INTERFACE I_NodePrototypes EXTENDS I_Serializable

METHOD PUBLIC InsertByType
VAR_INPUT
	NodeType : T_MAXSTRING;
	NodePrototype : I_NodePrototype;
END_VAR
END_METHOD

METHOD PUBLIC TryCreateByType : BOOL
VAR_INPUT
	NodeType : T_MAXSTRING;
	Destination : I_Node;
END_VAR
END_METHOD

END_INTERFACE

(* stored: Version 1.1.0.1, ProductVersion 3.1.4024.12
   Itf I_NodePrototypes: Id {f17dfa9a-d58a-0253-28a9-a9333d414dc7}
   Method InsertByType: Id {608f0d32-40ca-42da-a293-4636ec53d26a}
   Method TryCreateByType: Id {7791efde-3f8b-0c4c-15fc-4d13fe1c8d5a} *)
